   cmStackGripperFwdBwd.configuration.monitoringReachingFeedback := T#5S;
   cmStackGripperFwdBwd.configuration.monitoringDiscrepancy := T#0MS;
   cmStackGripperFwdBwd.configuration.setOutputHomeContinuously := TRUE;
   cmStackGripperFwdBwd.configuration.setOutputWorkContinuously := TRUE;
   cmStackGripperFwdBwd.configuration.disableHomeCommand := FALSE;
   cmStackGripperFwdBwd.configuration.disableFeedbackHomePos := FALSE;
   cmStackGripperFwdBwd.configuration.disableFeedbackWorkPos := FALSE;
   cmStackGripperFwdBwd.configuration.disableAlarms := FALSE;
   cmStackGripperFwdBwd.configuration.resetOutputsOnError := FALSE;
   cmStackGripperFwdBwd.configuration.allwaysWaitOnReachingTime := FALSE;
   cmJRWinderClampTopRearUpDown.commands.refreshConfiguration := FALSE;
   cmJRWinderClampTopRearUpDown.commands.editConfiguration := FALSE;
   cmJRWinderClampTopRearUpDown.commands.saveConfiguration := FALSE;
   cmJRWinderClampTopRearUpDown.commands.reset := FALSE;
   cmJRWinderClampTopRearUpDown.commands.commandHomePos := FALSE;
   cmJRWinderClampTopRearUpDown.commands.commandWorkPos := FALSE;
   cmJRWinderClampTopRearUpDown.monitoring.enable := TRUE;
   cmJRWinderClampTopRearUpDown.monitoring.referenceDesignator := WSTRING#'JRClampTopRearUpDown.';
   cmJRWinderClampTopRearUpDown.monitoring.commandHomePos := FALSE;
   cmJRWinderClampTopRearUpDown.monitoring.commandWorkPos := FALSE;
   cmJRWinderClampTopRearUpDown.monitoring.goToHomePos := TRUE;
   cmJRWinderClampTopRearUpDown.monitoring.goToWorkPos := FALSE;
   cmJRWinderClampTopRearUpDown.monitoring.inHomePos := TRUE;
   cmJRWinderClampTopRearUpDown.monitoring.inWorkPos := FALSE;
   cmJRWinderClampTopRearUpDown.monitoring.reset := FALSE;
   cmJRWinderClampTopRearUpDown.monitoring.enableManualCmds := FALSE;
   cmJRWinderClampTopRearUpDown.monitoring.error := FALSE;
   cmJRWinderClampTopRearUpDown.monitoring.interlockHomePos := TRUE;
   cmJRWinderClampTopRearUpDown.monitoring.interlockWorkPos := FALSE;
   cmJRWinderClampTopRearUpDown.monitoring.status := 16#7101;
   cmJRWinderClampTopRearUpDown.monitoring.interlockWarningWorkPos := FALSE;
   cmJRWinderClampTopRearUpDown.monitoring.interlockWarningHomePos := FALSE;
   cmJRWinderClampTopRearUpDown.configuration.referenceDesignator := WSTRING#'TwoWayAct.';
   cmJRWinderClampTopRearUpDown.configuration.monitoringLeavingFeedback := T#5S;
   cmJRWinderClampTopRearUpDown.configuration.monitoringReachingFeedback := T#5S;
   cmJRWinderClampTopRearUpDown.configuration.monitoringDiscrepancy := T#0MS;
   cmJRWinderClampTopRearUpDown.configuration.setOutputHomeContinuously := TRUE;
   cmJRWinderClampTopRearUpDown.configuration.setOutputWorkContinuously := TRUE;
   cmJRWinderClampTopRearUpDown.configuration.disableHomeCommand := FALSE;
   cmJRWinderClampTopRearUpDown.configuration.disableFeedbackHomePos := FALSE;
   cmJRWinderClampTopRearUpDown.configuration.disableFeedbackWorkPos := FALSE;
   cmJRWinderClampTopRearUpDown.configuration.disableAlarms := FALSE;
   cmJRWinderClampTopRearUpDown.configuration.resetOutputsOnError := FALSE;
   cmJRWinderClampTopRearUpDown.configuration.allwaysWaitOnReachingTime := FALSE;
   cmJRWinderClampBtmRearUpDown.commands.refreshConfiguration := FALSE;
   cmJRWinderClampBtmRearUpDown.commands.editConfiguration := FALSE;
   cmJRWinderClampBtmRearUpDown.commands.saveConfiguration := FALSE;
   cmJRWinderClampBtmRearUpDown.commands.reset := FALSE;
   cmJRWinderClampBtmRearUpDown.commands.commandHomePos := FALSE;
   cmJRWinderClampBtmRearUpDown.commands.commandWorkPos := FALSE;
   cmJRWinderClampBtmRearUpDown.monitoring.enable := TRUE;
   cmJRWinderClampBtmRearUpDown.monitoring.referenceDesignator := WSTRING#'JRClampBtmRearUpDown.';
   cmJRWinderClampBtmRearUpDown.monitoring.commandHomePos := FALSE;
   cmJRWinderClampBtmRearUpDown.monitoring.commandWorkPos := FALSE;
   cmJRWinderClampBtmRearUpDown.monitoring.goToHomePos := TRUE;
   cmJRWinderClampBtmRearUpDown.monitoring.goToWorkPos := FALSE;
   cmJRWinderClampBtmRearUpDown.monitoring.inHomePos := TRUE;
   cmJRWinderClampBtmRearUpDown.monitoring.inWorkPos := FALSE;
   cmJRWinderClampBtmRearUpDown.monitoring.reset := FALSE;
   cmJRWinderClampBtmRearUpDown.monitoring.enableManualCmds := FALSE;
   cmJRWinderClampBtmRearUpDown.monitoring.error := FALSE;
   cmJRWinderClampBtmRearUpDown.monitoring.interlockHomePos := TRUE;
   cmJRWinderClampBtmRearUpDown.monitoring.interlockWorkPos := TRUE;
   cmJRWinderClampBtmRearUpDown.monitoring.status := 16#7004;
   cmJRWinderClampBtmRearUpDown.monitoring.interlockWarningWorkPos := FALSE;
   cmJRWinderClampBtmRearUpDown.monitoring.interlockWarningHomePos := FALSE;
   cmJRWinderClampBtmRearUpDown.configuration.referenceDesignator := WSTRING#'JRClampBtmRearUpDown.';
   cmJRWinderClampBtmRearUpDown.configuration.monitoringLeavingFeedback := T#5S;
   cmJRWinderClampBtmRearUpDown.configuration.monitoringReachingFeedback := T#5S;
   cmJRWinderClampBtmRearUpDown.configuration.monitoringDiscrepancy := T#0MS;
   cmJRWinderClampBtmRearUpDown.configuration.setOutputHomeContinuously := TRUE;
   cmJRWinderClampBtmRearUpDown.configuration.setOutputWorkContinuously := TRUE;
   cmJRWinderClampBtmRearUpDown.configuration.disableHomeCommand := FALSE;
   cmJRWinderClampBtmRearUpDown.configuration.disableFeedbackHomePos := FALSE;
   cmJRWinderClampBtmRearUpDown.configuration.disableFeedbackWorkPos := FALSE;
   cmJRWinderClampBtmRearUpDown.configuration.disableAlarms := FALSE;
   cmJRWinderClampBtmRearUpDown.configuration.resetOutputsOnError := FALSE;
   cmJRWinderClampBtmRearUpDown.configuration.allwaysWaitOnReachingTime := FALSE;
   cmJRWinderClampTopFrontUpDown.commands.refreshConfiguration := FALSE;
   cmJRWinderClampTopFrontUpDown.commands.editConfiguration := FALSE;
   cmJRWinderClampTopFrontUpDown.commands.saveConfiguration := FALSE;
   cmJRWinderClampTopFrontUpDown.commands.reset := FALSE;
   cmJRWinderClampTopFrontUpDown.commands.commandHomePos := FALSE;
   cmJRWinderClampTopFrontUpDown.commands.commandWorkPos := FALSE;
   cmJRWinderClampTopFrontUpDown.monitoring.enable := TRUE;
   cmJRWinderClampTopFrontUpDown.monitoring.referenceDesignator := WSTRING#'JRClampTopFrontUpDown.';
   cmJRWinderClampTopFrontUpDown.monitoring.commandHomePos := FALSE;
   cmJRWinderClampTopFrontUpDown.monitoring.commandWorkPos := FALSE;
   cmJRWinderClampTopFrontUpDown.monitoring.goToHomePos := TRUE;
   cmJRWinderClampTopFrontUpDown.monitoring.goToWorkPos := FALSE;
   cmJRWinderClampTopFrontUpDown.monitoring.inHomePos := TRUE;
   cmJRWinderClampTopFrontUpDown.monitoring.inWorkPos := FALSE;
   cmJRWinderClampTopFrontUpDown.monitoring.reset := FALSE;
   cmJRWinderClampTopFrontUpDown.monitoring.enableManualCmds := FALSE;
   cmJRWinderClampTopFrontUpDown.monitoring.error := FALSE;
   cmJRWinderClampTopFrontUpDown.monitoring.interlockHomePos := TRUE;
   cmJRWinderClampTopFrontUpDown.monitoring.interlockWorkPos := TRUE;
   cmJRWinderClampTopFrontUpDown.monitoring.status := 16#7004;
   cmJRWinderClampTopFrontUpDown.monitoring.interlockWarningWorkPos := FALSE;
   cmJRWinderClampTopFrontUpDown.monitoring.interlockWarningHomePos := FALSE;
   cmJRWinderClampTopFrontUpDown.configuration.referenceDesignator := WSTRING#'JRClampTopFrontUpDown.';
   cmJRWinderClampTopFrontUpDown.configuration.monitoringLeavingFeedback := T#5S;
   cmJRWinderClampTopFrontUpDown.configuration.monitoringReachingFeedback := T#5S;
   cmJRWinderClampTopFrontUpDown.configuration.monitoringDiscrepancy := T#0MS;
   cmJRWinderClampTopFrontUpDown.configuration.setOutputHomeContinuously := TRUE;
   cmJRWinderClampTopFrontUpDown.configuration.setOutputWorkContinuously := TRUE;
   cmJRWinderClampTopFrontUpDown.configuration.disableHomeCommand := FALSE;
   cmJRWinderClampTopFrontUpDown.configuration.disableFeedbackHomePos := FALSE;
   cmJRWinderClampTopFrontUpDown.configuration.disableFeedbackWorkPos := FALSE;
   cmJRWinderClampTopFrontUpDown.configuration.disableAlarms := FALSE;
   cmJRWinderClampTopFrontUpDown.configuration.resetOutputsOnError := FALSE;
   cmJRWinderClampTopFrontUpDown.configuration.allwaysWaitOnReachingTime := FALSE;
   cmJRWinderClampBtmFrontUpDown.commands.refreshConfiguration := FALSE;
   cmJRWinderClampBtmFrontUpDown.commands.editConfiguration := FALSE;
   cmJRWinderClampBtmFrontUpDown.commands.saveConfiguration := FALSE;
   cmJRWinderClampBtmFrontUpDown.commands.reset := FALSE;
   cmJRWinderClampBtmFrontUpDown.commands.commandHomePos := FALSE;
   cmJRWinderClampBtmFrontUpDown.commands.commandWorkPos := FALSE;
   cmJRWinderClampBtmFrontUpDown.monitoring.enable := TRUE;
   cmJRWinderClampBtmFrontUpDown.monitoring.referenceDesignator := WSTRING#'JRClampBtmFrontUpDown.';
   cmJRWinderClampBtmFrontUpDown.monitoring.commandHomePos := FALSE;
   cmJRWinderClampBtmFrontUpDown.monitoring.commandWorkPos := FALSE;
   cmJRWinderClampBtmFrontUpDown.monitoring.goToHomePos := TRUE;
   cmJRWinderClampBtmFrontUpDown.monitoring.goToWorkPos := FALSE;
   cmJRWinderClampBtmFrontUpDown.monitoring.inHomePos := TRUE;
   cmJRWinderClampBtmFrontUpDown.monitoring.inWorkPos := FALSE;
   cmJRWinderClampBtmFrontUpDown.monitoring.reset := FALSE;
   cmJRWinderClampBtmFrontUpDown.monitoring.enableManualCmds := FALSE;
   cmJRWinderClampBtmFrontUpDown.monitoring.error := FALSE;
   cmJRWinderClampBtmFrontUpDown.monitoring.interlockHomePos := TRUE;
   cmJRWinderClampBtmFrontUpDown.monitoring.interlockWorkPos := TRUE;
   cmJRWinderClampBtmFrontUpDown.monitoring.status := 16#7004;
   cmJRWinderClampBtmFrontUpDown.monitoring.interlockWarningWorkPos := FALSE;
   cmJRWinderClampBtmFrontUpDown.monitoring.interlockWarningHomePos := FALSE;
   cmJRWinderClampBtmFrontUpDown.configuration.referenceDesignator := WSTRING#'JRClampBtmFrontUpDown.';
   cmJRWinderClampBtmFrontUpDown.configuration.monitoringLeavingFeedback := T#5S;
   cmJRWinderClampBtmFrontUpDown.configuration.monitoringReachingFeedback := T#5S;
   cmJRWinderClampBtmFrontUpDown.configuration.monitoringDiscrepancy := T#0MS;
   cmJRWinderClampBtmFrontUpDown.configuration.setOutputHomeContinuously := TRUE;
   cmJRWinderClampBtmFrontUpDown.configuration.setOutputWorkContinuously := TRUE;
   cmJRWinderClampBtmFrontUpDown.configuration.disableHomeCommand := FALSE;
   cmJRWinderClampBtmFrontUpDown.configuration.disableFeedbackHomePos := FALSE;
   cmJRWinderClampBtmFrontUpDown.configuration.disableFeedbackWorkPos := FALSE;
   cmJRWinderClampBtmFrontUpDown.configuration.disableAlarms := FALSE;
   cmJRWinderClampBtmFrontUpDown.configuration.resetOutputsOnError := FALSE;
   cmJRWinderClampBtmFrontUpDown.configuration.allwaysWaitOnReachingTime := FALSE;
   cmPusherRollerUpDown.commands.refreshConfiguration := FALSE;
   cmPusherRollerUpDown.commands.editConfiguration := FALSE;
   cmPusherRollerUpDown.commands.saveConfiguration := FALSE;
   cmPusherRollerUpDown.commands.reset := FALSE;
   cmPusherRollerUpDown.commands.commandHomePos := FALSE;
   cmPusherRollerUpDown.commands.commandWorkPos := FALSE;
   cmPusherRollerUpDown.monitoring.enable := FALSE;
   cmPusherRollerUpDown.monitoring.referenceDesignator := WSTRING#'PusherRollerUpDown';
   cmPusherRollerUpDown.monitoring.commandHomePos := FALSE;
   cmPusherRollerUpDown.monitoring.commandWorkPos := FALSE;
   cmPusherRollerUpDown.monitoring.goToHomePos := FALSE;
   cmPusherRollerUpDown.monitoring.goToWorkPos := FALSE;
   cmPusherRollerUpDown.monitoring.inHomePos := FALSE;
   cmPusherRollerUpDown.monitoring.inWorkPos := FALSE;
   cmPusherRollerUpDown.monitoring.reset := FALSE;
   cmPusherRollerUpDown.monitoring.enableManualCmds := FALSE;
   cmPusherRollerUpDown.monitoring.error := FALSE;
   cmPusherRollerUpDown.monitoring.interlockHomePos := FALSE;
   cmPusherRollerUpDown.monitoring.interlockWorkPos := FALSE;
   cmPusherRollerUpDown.monitoring.status := 16#0000;
   cmPusherRollerUpDown.monitoring.interlockWarningWorkPos := FALSE;
   cmPusherRollerUpDown.monitoring.interlockWarningHomePos := FALSE;
   cmPusherRollerUpDown.configuration.referenceDesignator := WSTRING#'PusherRollerUpDown';
   cmPusherRollerUpDown.configuration.monitoringLeavingFeedback := T#5S;
   cmPusherRollerUpDown.configuration.monitoringReachingFeedback := T#5S;
   cmPusherRollerUpDown.configuration.monitoringDiscrepancy := T#0MS;
   cmPusherRollerUpDown.configuration.setOutputHomeContinuously := TRUE;
   cmPusherRollerUpDown.configuration.setOutputWorkContinuously := TRUE;
   cmPusherRollerUpDown.configuration.disableHomeCommand := FALSE;
   cmPusherRollerUpDown.configuration.disableFeedbackHomePos := FALSE;
   cmPusherRollerUpDown.configuration.disableFeedbackWorkPos := FALSE;
   cmPusherRollerUpDown.configuration.disableAlarms := FALSE;
   cmPusherRollerUpDown.configuration.resetOutputsOnError := FALSE;
   cmPusherRollerUpDown.configuration.allwaysWaitOnReachingTime := FALSE;
   cmPusherRollerFwdBwd.commands.refreshConfiguration := FALSE;
   cmPusherRollerFwdBwd.commands.editConfiguration := FALSE;
   cmPusherRollerFwdBwd.commands.saveConfiguration := FALSE;
   cmPusherRollerFwdBwd.commands.reset := FALSE;
   cmPusherRollerFwdBwd.commands.commandHomePos := FALSE;
   cmPusherRollerFwdBwd.commands.commandWorkPos := FALSE;
   cmPusherRollerFwdBwd.monitoring.enable := TRUE;
   cmPusherRollerFwdBwd.monitoring.referenceDesignator := WSTRING#'PusherRollerFwdBwd';
   cmPusherRollerFwdBwd.monitoring.commandHomePos := FALSE;
   cmPusherRollerFwdBwd.monitoring.commandWorkPos := FALSE;
   cmPusherRollerFwdBwd.monitoring.goToHomePos := TRUE;
   cmPusherRollerFwdBwd.monitoring.goToWorkPos := FALSE;
   cmPusherRollerFwdBwd.monitoring.inHomePos := TRUE;
   cmPusherRollerFwdBwd.monitoring.inWorkPos := FALSE;
   cmPusherRollerFwdBwd.monitoring.reset := FALSE;
   cmPusherRollerFwdBwd.monitoring.enableManualCmds := FALSE;
   cmPusherRollerFwdBwd.monitoring.error := FALSE;
   cmPusherRollerFwdBwd.monitoring.interlockHomePos := TRUE;
   cmPusherRollerFwdBwd.monitoring.interlockWorkPos := TRUE;
   cmPusherRollerFwdBwd.monitoring.status := 16#7004;
   cmPusherRollerFwdBwd.monitoring.interlockWarningWorkPos := FALSE;
   cmPusherRollerFwdBwd.monitoring.interlockWarningHomePos := FALSE;
   cmPusherRollerFwdBwd.configuration.referenceDesignator := WSTRING#'PusherRollerFwdBwd';
   cmPusherRollerFwdBwd.configuration.monitoringLeavingFeedback := T#5S;
   cmPusherRollerFwdBwd.configuration.monitoringReachingFeedback := T#5S;
   cmPusherRollerFwdBwd.configuration.monitoringDiscrepancy := T#0MS;
   cmPusherRollerFwdBwd.configuration.setOutputHomeContinuously := TRUE;
   cmPusherRollerFwdBwd.configuration.setOutputWorkContinuously := TRUE;
   cmPusherRollerFwdBwd.configuration.disableHomeCommand := FALSE;
   cmPusherRollerFwdBwd.configuration.disableFeedbackHomePos := FALSE;
   cmPusherRollerFwdBwd.configuration.disableFeedbackWorkPos := FALSE;
   cmPusherRollerFwdBwd.configuration.disableAlarms := FALSE;
   cmPusherRollerFwdBwd.configuration.resetOutputsOnError := FALSE;
   cmPusherRollerFwdBwd.configuration.allwaysWaitOnReachingTime := FALSE;
   intCondition.Axis_34.Home.HomeInterlock := FALSE;
   intCondition.Axis_34.Home.homeinterlock_error := FALSE;
   intCondition.Axis_34.Home.intout[0..9] := FALSE;
   intCondition.Axis_34.Jog.ForwardInterlockOK := FALSE;
   intCondition.Axis_34.Jog.BackwardInterlockOk := FALSE;
   intCondition.Axis_34.Jog.ForwardInterlockError := FALSE;
   intCondition.Axis_34.Jog.BackwardInterlockError := FALSE;
   intCondition.Axis_34.Jog.intOut[0..9] := FALSE;
   intCondition.Axis_34.Position.interlockOk[0..15] := FALSE;
   intCondition.Axis_34.Position.interlockError[0..15] := FALSE;
   intCondition.Axis_34.Position.intOut[0..9] := FALSE;
   intCondition.Axis_35.Home.HomeInterlock := FALSE;
   intCondition.Axis_35.Home.homeinterlock_error := FALSE;
   intCondition.Axis_35.Home.intout[0..9] := FALSE;
   intCondition.Axis_35.Jog.ForwardInterlockOK := FALSE;
   intCondition.Axis_35.Jog.BackwardInterlockOk := FALSE;
   intCondition.Axis_35.Jog.ForwardInterlockError := FALSE;
   intCondition.Axis_35.Jog.BackwardInterlockError := FALSE;
   intCondition.Axis_35.Jog.intOut[0..9] := FALSE;
   intCondition.Axis_35.Position.interlockOk[0..15] := FALSE;
   intCondition.Axis_35.Position.interlockError[0..15] := FALSE;
   intCondition.Axis_35.Position.intOut[0..9] := FALSE;
   intCondition.Axis_36.Home.HomeInterlock := FALSE;
   intCondition.Axis_36.Home.homeinterlock_error := FALSE;
   intCondition.Axis_36.Home.intout[0..9] := FALSE;
   intCondition.Axis_36.Jog.ForwardInterlockOK := FALSE;
   intCondition.Axis_36.Jog.BackwardInterlockOk := FALSE;
   intCondition.Axis_36.Jog.ForwardInterlockError := FALSE;
   intCondition.Axis_36.Jog.BackwardInterlockError := FALSE;
   intCondition.Axis_36.Jog.intOut[0..9] := FALSE;
   intCondition.Axis_36.Position.interlockOk[0..15] := FALSE;
   intCondition.Axis_36.Position.interlockError[0..15] := FALSE;
   intCondition.Axis_36.Position.intOut[0..9] := FALSE;
   intCondition.Axis_37.Home.HomeInterlock := FALSE;
   intCondition.Axis_37.Home.homeinterlock_error := FALSE;
   intCondition.Axis_37.Home.intout[0..9] := FALSE;
   intCondition.Axis_37.Jog.ForwardInterlockOK := FALSE;
   intCondition.Axis_37.Jog.BackwardInterlockOk := FALSE;
   intCondition.Axis_37.Jog.ForwardInterlockError := FALSE;
   intCondition.Axis_37.Jog.BackwardInterlockError := FALSE;
   intCondition.Axis_37.Jog.intOut[0..9] := FALSE;
   intCondition.Axis_37.Position.interlockOk[0..15] := FALSE;
   intCondition.Axis_37.Position.interlockError[0..15] := FALSE;
   intCondition.Axis_37.Position.intOut[0..9] := FALSE;
   intCondition.Axis_38.Home.HomeInterlock := FALSE;
   intCondition.Axis_38.Home.homeinterlock_error := FALSE;
   intCondition.Axis_38.Home.intout[0..9] := FALSE;
   intCondition.Axis_38.Jog.ForwardInterlockOK := FALSE;
   intCondition.Axis_38.Jog.BackwardInterlockOk := FALSE;
   intCondition.Axis_38.Jog.ForwardInterlockError := FALSE;
   intCondition.Axis_38.Jog.BackwardInterlockError := FALSE;
   intCondition.Axis_38.Jog.intOut[0..9] := FALSE;
   intCondition.Axis_38.Position.interlockOk[0..15] := FALSE;
   intCondition.Axis_38.Position.interlockError[0..15] := FALSE;
   intCondition.Axis_38.Position.intOut[0..9] := FALSE;
   intCondition.Axis_39.Home.HomeInterlock := FALSE;
   intCondition.Axis_39.Home.homeinterlock_error := FALSE;
   intCondition.Axis_39.Home.intout[0..9] := FALSE;
   intCondition.Axis_39.Jog.ForwardInterlockOK := FALSE;
   intCondition.Axis_39.Jog.BackwardInterlockOk := FALSE;
   intCondition.Axis_39.Jog.ForwardInterlockError := FALSE;
   intCondition.Axis_39.Jog.BackwardInterlockError := FALSE;
   intCondition.Axis_39.Jog.intOut[0..9] := FALSE;
   intCondition.Axis_39.Position.interlockOk[0..15] := FALSE;
   intCondition.Axis_39.Position.interlockError[0..15] := FALSE;
   intCondition.Axis_39.Position.intOut[0..9] := FALSE;
   intCondition.Axis_40.Home.HomeInterlock := FALSE;
   intCondition.Axis_40.Home.homeinterlock_error := FALSE;
   intCondition.Axis_40.Home.intout[0..9] := FALSE;
   intCondition.Axis_40.Jog.ForwardInterlockOK := FALSE;
   intCondition.Axis_40.Jog.BackwardInterlockOk := FALSE;
   intCondition.Axis_40.Jog.ForwardInterlockError := FALSE;
   intCondition.Axis_40.Jog.BackwardInterlockError := FALSE;
   intCondition.Axis_40.Jog.intOut[0..9] := FALSE;
   intCondition.Axis_40.Position.interlockOk[0..15] := FALSE;
   intCondition.Axis_40.Position.interlockError[0..15] := FALSE;
   intCondition.Axis_40.Position.intOut[0..9] := FALSE;
   intCondition.Axis_41.Home.HomeInterlock := FALSE;
   intCondition.Axis_41.Home.homeinterlock_error := FALSE;
   intCondition.Axis_41.Home.intout[0..9] := FALSE;
   intCondition.Axis_41.Jog.ForwardInterlockOK := FALSE;
   intCondition.Axis_41.Jog.BackwardInterlockOk := FALSE;
   intCondition.Axis_41.Jog.ForwardInterlockError := FALSE;
   intCondition.Axis_41.Jog.BackwardInterlockError := FALSE;
   intCondition.Axis_41.Jog.intOut[0..9] := FALSE;
   intCondition.Axis_41.Position.interlockOk[0..15] := FALSE;
   intCondition.Axis_41.Position.interlockError[0..15] := FALSE;
   intCondition.Axis_41.Position.intOut[0..9] := FALSE;
   intCondition.Axis_42.Home.HomeInterlock := FALSE;
   intCondition.Axis_42.Home.homeinterlock_error := FALSE;
   intCondition.Axis_42.Home.intout[0..9] := FALSE;
   intCondition.Axis_42.Jog.ForwardInterlockOK := FALSE;
   intCondition.Axis_42.Jog.BackwardInterlockOk := FALSE;
   intCondition.Axis_42.Jog.ForwardInterlockError := FALSE;
   intCondition.Axis_42.Jog.BackwardInterlockError := FALSE;
   intCondition.Axis_42.Jog.intOut[0..9] := FALSE;
   intCondition.Axis_42.Position.interlockOk[0..15] := FALSE;
   intCondition.Axis_42.Position.interlockError[0..15] := FALSE;
   intCondition.Axis_42.Position.intOut[0..9] := FALSE;
   intCondition.Axis_04.Home.HomeInterlock := FALSE;
   intCondition.Axis_04.Home.homeinterlock_error := FALSE;
   intCondition.Axis_04.Home.intout[0..9] := FALSE;
   intCondition.Axis_04.Jog.ForwardInterlockOK := FALSE;
   intCondition.Axis_04.Jog.BackwardInterlockOk := FALSE;
   intCondition.Axis_04.Jog.ForwardInterlockError := FALSE;
   intCondition.Axis_04.Jog.BackwardInterlockError := FALSE;
   intCondition.Axis_04.Jog.intOut[0..9] := FALSE;
   intCondition.Axis_04.Position.interlockOk[0..15] := FALSE;
   intCondition.Axis_04.Position.interlockError[0..15] := FALSE;
   intCondition.Axis_04.Position.intOut[0..9] := FALSE;
   intCondition.Actuator_38.Home_INT := FALSE;
   intCondition.Actuator_38.Work_INT := FALSE;
   intCondition.Actuator_38.Home_INT_Error := FALSE;
   intCondition.Actuator_38.Work_INT_Error := FALSE;
   intCondition.Actuator_38.intOut[0..9] := FALSE;
   intCondition.Actuator_39.Home_INT := FALSE;
   intCondition.Actuator_39.Work_INT := FALSE;
   intCondition.Actuator_39.Home_INT_Error := FALSE;
   intCondition.Actuator_39.Work_INT_Error := FALSE;
   intCondition.Actuator_39.intOut[0..9] := FALSE;
   intCondition.Actuator_40.Home_INT := FALSE;
   intCondition.Actuator_40.Work_INT := FALSE;
   intCondition.Actuator_40.Home_INT_Error := FALSE;
   intCondition.Actuator_40.Work_INT_Error := FALSE;
   intCondition.Actuator_40.intOut[0..9] := FALSE;
   intCondition.Actuator_41.Home_INT := FALSE;
   intCondition.Actuator_41.Work_INT := FALSE;
   intCondition.Actuator_41.Home_INT_Error := FALSE;
   intCondition.Actuator_41.Work_INT_Error := FALSE;
   intCondition.Actuator_41.intOut[0..9] := FALSE;
   intCondition.Actuator_42.Home_INT := FALSE;
   intCondition.Actuator_42.Work_INT := FALSE;
   intCondition.Actuator_42.Home_INT_Error := FALSE;
   intCondition.Actuator_42.Work_INT_Error := FALSE;
   intCondition.Actuator_42.intOut[0..9] := FALSE;
   intCondition.Actuator_43.Home_INT := FALSE;
   intCondition.Actuator_43.Work_INT := FALSE;
   intCondition.Actuator_43.Home_INT_Error := FALSE;
   intCondition.Actuator_43.Work_INT_Error := FALSE;
   intCondition.Actuator_43.intOut[0..9] := FALSE;
   intCondition.Actuator_44.Home_INT := FALSE;
   intCondition.Actuator_44.Work_INT := FALSE;
   intCondition.Actuator_44.Home_INT_Error := FALSE;
   intCondition.Actuator_44.Work_INT_Error := FALSE;
   intCondition.Actuator_44.intOut[0..9] := FALSE;
   intCondition.Actuator_45.Home_INT := FALSE;
   intCondition.Actuator_45.Work_INT := FALSE;
   intCondition.Actuator_45.Home_INT_Error := FALSE;
   intCondition.Actuator_45.Work_INT_Error := FALSE;
   intCondition.Actuator_45.intOut[0..9] := FALSE;
   intCondition.Actuator_46.Home_INT := FALSE;
   intCondition.Actuator_46.Work_INT := FALSE;
   intCondition.Actuator_46.Home_INT_Error := FALSE;
   intCondition.Actuator_46.Work_INT_Error := FALSE;
   intCondition.Actuator_46.intOut[0..9] := FALSE;
   intCondition.Actuator_47.Home_INT := FALSE;
   intCondition.Actuator_47.Work_INT := FALSE;
   intCondition.Actuator_47.Home_INT_Error := FALSE;
   intCondition.Actuator_47.Work_INT_Error := FALSE;
   intCondition.Actuator_47.intOut[0..9] := FALSE;
   intCondition.Actuator_48.Home_INT := FALSE;
   intCondition.Actuator_48.Work_INT := FALSE;
   intCondition.Actuator_48.Home_INT_Error := FALSE;
   intCondition.Actuator_48.Work_INT_Error := FALSE;
   intCondition.Actuator_48.intOut[0..9] := FALSE;
   intCondition.Actuator_49.Home_INT := FALSE;
   intCondition.Actuator_49.Work_INT := FALSE;
   intCondition.Actuator_49.Home_INT_Error := FALSE;
   intCondition.Actuator_49.Work_INT_Error := FALSE;
   intCondition.Actuator_49.intOut[0..9] := FALSE;
END_DATA_BLOCK
